// TwinCAT 3 PLC project StringsTest
// ProgramVersion: 3.1.4024.0
// libraries:
//   Strings, * (TomasRompotl)
//   Tc2_System, * (Beckhoff Automation GmbH)
//   Tc3_Module, * (Beckhoff Automation GmbH)
//   TcUnit, * (www.tcunit.org)
//   Types, * (TomasRompotl)
// project tree:
//   Builders/ BuildStringInlineTest.TcPOU (not stored), StringBuilder255Test.TcPOU (not stored), StringBuilderExtBufferTest.TcPOU (not stored), StringBuilderInfiniteTest.TcPOU (not stored)
//   Convert/ ConvertFunctionsTest.TcPOU (not stored)
//   Manipulate/ ManipulateFunctionsTest.TcPOU (not stored)
//   / PlcTask.TcTTO, PRG_Test.TcPOU
//   Validate/ ValidateFunctionsTest.TcPOU
// (motion and I/O tree: see PLC project typestest)
// real-time tasks:
//   TASK TypesTestTask: cycle T#1ms, priority 20, ADS port 350
//   TASK StringsTestTask: cycle T#1ms, priority 21, ADS port 351
//   TASK DataTestTask: cycle T#1ms, priority 22, ADS port 352
//   TASK MathTestTask: cycle T#1ms, priority 23, ADS port 353
//   TASK TimesTestTask: cycle T#1ms, priority 24, ADS port 354

CONFIGURATION StringsTest
    RESOURCE PLC ON TwinCAT3
        TASK PlcTask(INTERVAL := T#1ms, PRIORITY := 21);
        PROGRAM PRG_Test WITH PlcTask : PRG_Test;
    END_RESOURCE
END_CONFIGURATION

// ---- PRG_Test.TcPOU
PROGRAM PRG_Test
VAR
	validateFunctionsTest : ValidateFunctionsTest;
	manipulateFunctionsTest : ManipulateFunctionsTest;
	convertFunctionsTest : ConvertFunctionsTest;
	
	sb255Test : StringBuilder255Test;
	buildStringInlineTest : BuildStringInlineTest;
	sbExtBufferTest : StringBuilderExtBufferTest;
	sbInfiniteTest : StringBuilderInfiniteTest;
END_VAR

TcUnit.RUN();

END_PROGRAM

// ---- Validate/ValidateFunctionsTest.TcPOU
FUNCTION_BLOCK ValidateFunctionsTest EXTENDS TcUnit.FB_TestSuite
VAR
END_VAR

StringBeginsWithAnyFunction();
StringEndsWithAnyFunction();

METHOD StringBeginsWithAnyFunction : BOOL
VAR
	test : T_MaxString := 'this is test string';
END_VAR
TcUnit.TEST('String begins with');

AssertEquals_BOOL(
	Expected := FALSE,
	Actual := StringBeginsWithAny(test, 'nothing'),
	Message := 'Should return FALSE because string does not begin with checked value');

AssertEquals_BOOL(
	Expected := TRUE,
	Actual := StringBeginsWithAny(test, 'this'),
	Message := 'Should return TRUE because string begins with checked value');

TEST_FINISHED();
END_METHOD

METHOD StringEndsWithAnyFunction : BOOL
VAR
	test : T_MaxString := 'this is test string';
END_VAR
TcUnit.TEST('String ends with');

AssertEquals_BOOL(
	Expected := FALSE,
	Actual := StringBeginsWithAny(test, 'nothing'),
	Message := 'Should return FALSE because string does not end with checked value');

AssertEquals_BOOL(
	Expected := TRUE,
	Actual := StringEndsWithAny(test, 'string'),
	Message := 'Should return TRUE because string ends with checked value');

TEST_FINISHED();
END_METHOD

END_FUNCTION_BLOCK
